TYPE ST_Analytics :
STRUCT
	nUnitsProduced : ULINT;
	nDefectiveUnits : ULINT;
	nState : UINT;
	tMlCalculation : TIME;
	bDefectivePart : BOOL;
END_STRUCT
END_TYPE

(* stored: Version 1.1.0.1, ProductVersion 3.1.4024.13
   DUT ST_Analytics: Id {3a8cb4dd-2be7-4941-b03f-24e457815e17} *)
